ABB RobotStudio station: 2_0P4_pokorny_20200416-211753.rsstn

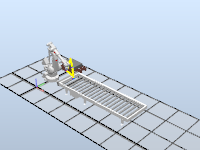
Station 2_0P4_pokorny (saved by RobotStudio 7.0.8743.626)
Controller Controller1, task T_ROB1: task frame (RAPID world) sits at (0, 1000, 0) mm in the station
Controller Controller1
  mechanical unit ROB_1: IRB4400_60_196__03, 6 joints, base frame (0, 0, 0) mm
Layout (positions relative to the parent item):
  - IRB4400_60_196__03 [mechanism, from Robots\IRB4400_60_196_G_03.rslib] at (0, 1000, 0) mm; joint values [0, 0.0631, 0.5639, 0, 1.0069, 0] (rad or m)
  - 1200_4000_h2_conveyor [part, from Equipment\Conveyor 1200 4000 h2.rslib] at (1000, 600, 0) mm
  - vac_gripper [mechanism] at (1080, 1000, 1084.64) mm, rotated rx 180 ry 0 rz 180 deg
      TCP vac_gripper at (0, 0, 176.61) mm
      links: gripper
  - Euro Pallet [graphiccomponentgroup, from Equipment\Euro Pallet.rslib] at (-600, 2000, 0) mm
    - Body 1 [part, from Equipment\Euro Pallet.rslib]
  - box_1 [part, from Libraries\box_1.rslib] at (1200, 1000, 415) mm
  - Positioner [smart component, from Components\Positioner.rslib]
      properties: Object=box_1; Position=[1.2 1 0.415]; Orientation=[0 0 0]; Reference=Global; ReferenceObject=(none)
  - box_1_2 [part, from Libraries\box_1.rslib] at (-600, 2500, 145) mm
  - Attacher [smart component, from Components\Attacher.rslib] at (0, 1000, 0) mm
      properties: Parent=vac_gripper; Flange=0; Child=box_1_92; Mount=false; Offset=[0 0 0]; Orientation=[0 0 0]
  - Detacher [smart component, from Components\Detacher.rslib]
      properties: Child=box_1_92; KeepPosition=true
  - box_conv [part, from Libraries\box_1.rslib] at (4200, 1000, 415) mm
  - Source_3 [smart component, from Components\Source.rslib]
      properties: Source=box_1; Copy=box_1_92; Parent=(none); Position=[1.2 1 0.415]; Orientation=[0 0 0]; Transient=false; PhysicsBehavior=0
  - box_1_87 [part, from Libraries\box_1.rslib] at (-600, 2500, 145) mm
  - box_1_88 [part, from Libraries\box_1.rslib] at (-300, 2500, 145) mm
  - box_1_89 [part, from Libraries\box_1.rslib] at (0, 2500, 145) mm
  - box_1_90 [part, from Libraries\box_1.rslib] at (-600, 2200, 145) mm
  - box_1_91 [part, from Libraries\box_1.rslib] at (-300, 2200, 145) mm
  - box_1_92 [part, from Libraries\box_1.rslib] at (0, 2200, 145) mm
  - Frame_1 [frame] at (0, 0, 176.61) mm
Attachment: vac_gripper is attached to IRB4400_60_196__03 / Link6
Attachment: Attacher is attached to IRB4400_60_196__03 / Base
Station signals: DI box_1_positioner, DI spawn_box
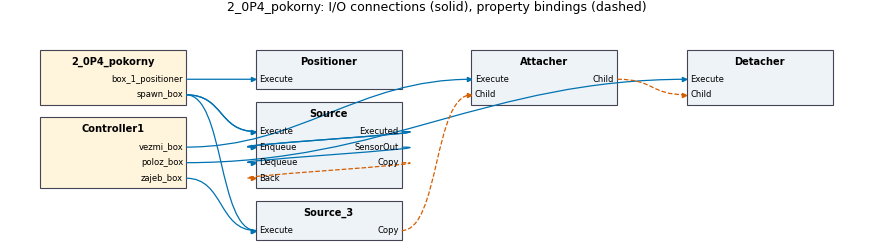
Station logic (signal -> signal, property => property):
  2_0P4_pokorny.box_1_positioner -> Positioner.Execute
  Controller1.vezmi_box -> Attacher.Execute
  Controller1.poloz_box -> Detacher.Execute
  2_0P4_pokorny.spawn_box -> Source.Execute
  Source.Executed -> Queue.Enqueue
  PlaneSensor.SensorOut -> Queue.Dequeue
  2_0P4_pokorny.spawn_box -> Source_2.Execute
  Source_2.Executed -> Queue.Enqueue
  2_0P4_pokorny.spawn_box -> Source_3.Execute
  Controller1.zajeb_box -> Source_3.Execute
  Source.Copy => Queue.Back
  Source_3.Copy => Attacher.Child
  Attacher.Child => Detacher.Child
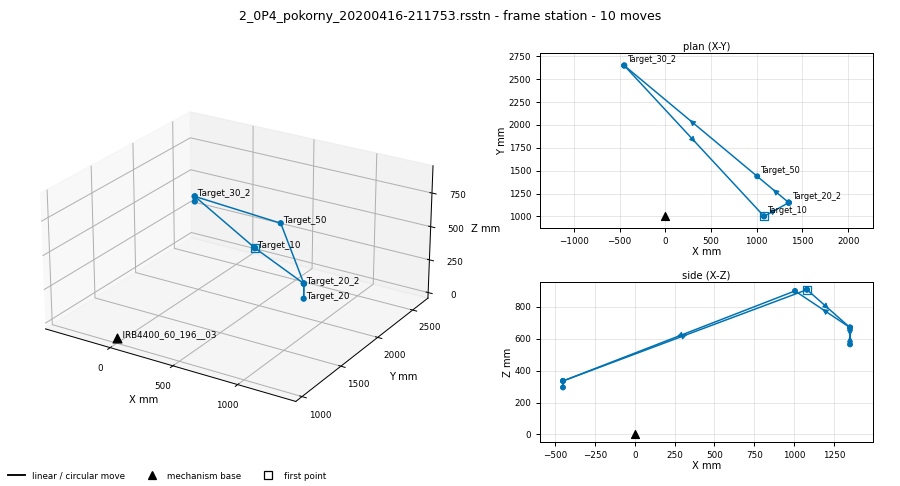
[picture p0: tool path of 2_0P4_pokorny_20200416-211753.rsstn in frame station, 10 of 10 moves have a stored position in this frame; points joined in program order, loops and branches not executed]
Targets, tools, work objects and paths stored in the station, written as RAPID:
! task T_ROB1
MODULE Module1
  CONST robtarget Target_10:=[[1080,0,908.028317799],[0,0,1,0],[0,0,0,0],[9E+09,9E+09,9E+09,9E+09,9E+09,9E+09]];
  CONST robtarget Target_20:=[[1350,150,565],[0,0,1,0],[0,0,0,0],[9E+09,9E+09,9E+09,9E+09,9E+09,9E+09]];
  CONST robtarget Target_20_2:=[[1350,150,670.31163825],[0,0,1,0],[0,0,0,0],[9E+09,9E+09,9E+09,9E+09,9E+09,9E+09]];
  CONST robtarget Target_30:=[[-450,1650,295],[0,0,1,0],[1,0,1,0],[9E+09,9E+09,9E+09,9E+09,9E+09,9E+09]];
  CONST robtarget Target_30_2:=[[-450,1650,335.435889427],[0,0,1,0],[1,0,1,0],[9E+09,9E+09,9E+09,9E+09,9E+09,9E+09]];
  CONST robtarget Target_40:=[[1004.829998529,437.649980689,899.999994623],[-0.00000002,0,1,-0.000000009],[0,-1,0,0],[9E+09,9E+09,9E+09,9E+09,9E+09,9E+09]];
  CONST robtarget Target_50:=[[1004.83,437.65,900],[0,0,1,0],[0,0,0,0],[9E+09,9E+09,9E+09,9E+09,9E+09,9E+09]];
  PROC Path_10()
    PulseDO zajeb_box;
    MoveL Target_10,v1000,z100,vac_gripper\WObj:=wobj0;
    MoveL Target_20_2,v1000,fine,vac_gripper\WObj:=wobj0;
    MoveL Target_20_2,v500,z100,vac_gripper\WObj:=wobj0;
    MoveL Target_20,v300,fine,vac_gripper\WObj:=wobj0;
    PulseDO vezmi_box;
    WaitTime 1;
    MoveL Target_20_2,v1000,fine,vac_gripper\WObj:=wobj0;
    MoveL Target_50,v1000,z200,vac_gripper\WObj:=wobj0;
    MoveL Target_30_2,v1000,z100,vac_gripper\WObj:=wobj0;
    MoveL Target_30,v300,fine,vac_gripper\WObj:=wobj0;
    PulseDO poloz_box;
    WaitTime 1;
    MoveL Target_30_2,v1000,fine,vac_gripper\WObj:=wobj0;
    MoveL Target_10,v2000,z100,vac_gripper\WObj:=wobj0;
  ENDPROC
  PROC main()
    Path_10;
  ENDPROC
ENDMODULE

! task T_ROB1
MODULE CalibData
  PERS tooldata vac_gripper:=[TRUE,[[0,0,176.61],[1,0,0,0]],[1,[0,0,50.915],[1,0,0,0],0,0,0]];
ENDMODULE

